PROGRAM MAIN
VAR
	nCounter: INT;
END_VAR

//

nCounter := nCounter + 1;

ACTION ACT_deneme:

END_ACTION

END_PROGRAM

(* stored: Version 1.1.0.1, ProductVersion 3.1.4024.15
   POU MAIN: Id {4ed37e00-bb03-4a14-80ff-f38f7977a9e4}, SpecialFunc None
   Action ACT_deneme: Id {6305d8ff-c27a-49cd-8dfc-08fba6290b48} *)
